(* PLC project Unnamed, Unknown Unnamed 1 *)
(* stored: creationDateTime 2016-12-29T13:37:46, modificationDateTime 2017-01-19T00:25:21 *)

PROGRAM program0
  VAR
    LocalVar0 : INT;
  END_VAR

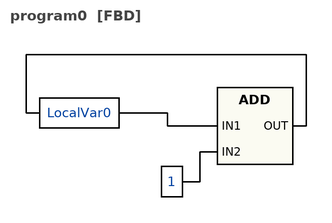
(* FBD diagram, written out as Structured Text *)
LocalVar0 := LocalVar0 + 1;
END_PROGRAM

CONFIGURATION config
  RESOURCE resource1 ON PLC
    TASK task_1(INTERVAL := T#1ms, PRIORITY := 0);
    PROGRAM inst_1 WITH task_1 : program0;
  END_RESOURCE
END_CONFIGURATION
